{attribute 'qualified_only'}
VAR_GLOBAL
//Przyciski zmaiany stanu	
//	fbprUndefined			: FB_RequestChanges;
	fbprAbort				: FB_IOButton_NO;
  	fbprClear				: FB_IOButton_NO;
   	fbprReset				: FB_IOButton_NO;
   	fbprStart				: FB_IOButton_NO;
   	fbprStop				: FB_IOButton_NO;
   	fbprHold				: FB_IOButton_NO;
   	fbprUnhold				: FB_IOButton_NO;
   	fbprSuspend				: FB_IOButton_NO;
   	fbprUnsuspend			: FB_IOButton_NO;
  	fbprComplete			: FB_IOButton_NO;
//przyciski zmiany trybu
//	fbprNiedozwolony		: FB_SITP_PolecenieZmianyTrybu (ePolecenie := E_SITP_PolecenieZmianyTrybu.brak);     
	fbprProduction			: FB_IOButton_NO;
    fbprMaintenance			: FB_IOButton_NO;
    fbprManual				: FB_IOButton_NO;
    fbprWashing				: FB_IOButton_NO;
    fbprDiagnostics			: FB_IOButton_NO;
//    fbprUzytkownika2		: FB_RequestChanges;
//   fbprUzytkownika3		: FB_RequestChanges;
//    fbprUzytkownika4		: FB_RequestChanges;
//    fbprUzytkownika5		: FB_RequestChanges;

END_VAR

(* stored: Version 1.1.0.1
   GVL GVL_RequeestChange: Id {70707167-7928-09eb-357f-a2f4dc4e8a35} *)
